// TIA Portal V17 export
// export: Created 2023-12-22T15:28:38.0396154Z, ExportSetting WithDefaults, DisplayName Totally Integrated Automation Portal, DisplayVersion V17, DisplayName TIA Portal Openness, DisplayVersion V17, DisplayName TIA Portal Version Control Interface, DisplayVersion V17, DisplayName STEP 7 Professional, DisplayVersion V17, DisplayName STEP 7 Safety, DisplayVersion V17, DisplayName WinCC Advanced, DisplayVersion V17
VAR_GLOBAL   // PLC tag table "System_Tags"
   pulse_01s AT %M10.0 : Bool;
   pulse_05s AT %M10.1 : Bool;
   pulse_1s AT %M10.2 : Bool;
   pulse_5s AT %M10.3 : Bool;
   pulse_10s AT %M10.4 : Bool;
   pulse_30s AT %M10.5 : Bool;
   pulse_1m AT %M10.6 : Bool;
   pulse_5m AT %M10.7 : Bool;
   pulse_10m AT %M11.0 : Bool;
   pulse_1h AT %M11.2 : Bool;
   TRUE AT %M1.2 : Bool;
   FALSE AT %M1.3 : Bool;
   Hand_DI AT %M12.0 : Bool;
   Hand_DO AT %M12.1 : Bool;
   Hand_AI AT %M12.2 : Bool;
   Hand_AO AT %M12.3 : Bool;
   Hand_M AT %M12.4 : Bool;
   Hand_MD AT %M12.5 : Bool;
   Hand_MDA AT %M12.6 : Bool;
   Hand_V AT %M12.7 : Bool;
   Hand_VD2 AT %M13.0 : Bool;
   Hand_VDA AT %M13.1 : Bool;
   Hand_Any AT %M13.7 : Bool;
   Alm_AI AT %M14.0 : Bool;
   Alm_M AT %M14.1 : Bool;
   Alm_MD AT %M14.2 : Bool;
   Alm_MDA AT %M14.3 : Bool;
   Alm_V AT %M14.4 : Bool;
   Alm_VD2 AT %M14.5 : Bool;
   Alm_VDA AT %M14.6 : Bool;
   Alm_Logick AT %M14.7 : Bool;
   Alm_Any AT %M15.7 : Bool;
   All_Block AT %M2.0 : Bool;
   Reset_All AT %M3.0 : Bool;
   Local_Mode AT %M4.0 : Bool;
   Sim_All AT %M5.0 : Bool;
   AI_Val_1 AT %MB100 : Byte;
   AI_Val_2 AT %MB101 : Byte;
   AI_Value AT %MW100 : Word;
   AO_Val_1 AT %MB102 : Byte;
   AO_Val_2 AT %MB103 : Byte;
   AO_Value AT %MW102 : Word;
   Events AT %MW200 : Word;
   pulse_1_day AT %M11.3 : Bool;
   pulse_1_week AT %M11.4 : Bool;
   pulse_1_month AT %M11.5 : Bool;
   pulse_30m AT %M11.1 : Bool;
   pulse_s1 AT %M11.6 : Bool;
   pulse_s2 AT %M11.7 : Bool;
   Hand_Low AT %M13.5 : Bool;
   Hand_High AT %M13.6 : Bool;
   Reset_Hand AT %M3.1 : Bool;
   Events_pos AT %MW210 : Word;
   Alarms AT %MW202 : Word;
   Alarms_pos AT %MW212 : Word;
END_VAR
